FUNCTION_BLOCK PUBLIC FB_FinalTest

VAR
	
END_VAR

METHOD FB_Opto22Read : BOOL
VAR_INPUT
END_VAR
END_METHOD

METHOD FB_Opto22Write : BOOL
VAR_INPUT
END_VAR
END_METHOD

METHOD PUBLIC LeakTest : BOOL
VAR_INPUT
END_VAR
END_METHOD

METHOD PRIVATE ModuleCheck : BOOL
VAR_INPUT
END_VAR
END_METHOD

END_FUNCTION_BLOCK

(* stored: Version 1.1.0.1, ProductVersion 3.1.4024.9
   POU FB_FinalTest: Id {f7c9b199-23a8-4316-8294-e5afe3220f77}, SpecialFunc None
   Method FB_Opto22Read: Id {7dc0df06-147c-4ee3-b374-8c9ccca4d543}
   Method FB_Opto22Write: Id {79f7331f-4009-4dec-8020-ef05673366f1}
   Method LeakTest: Id {263c8cfe-7a2f-4231-b3e4-7f002a5e9e71}
   Method ModuleCheck: Id {c89c3e22-89a6-41b9-b0f5-144d51810253} *)
